// TIA Portal V18 export
DATA_BLOCK "Timers_DB"   // DB21
// stored: AutoNumber false, InstanceOfName Timers, InstanceOfType FB
"Timers"
   // VAR
   //    TDTimeReset : Bool;
   //    M1TimeReset : Bool;
   //    M2TimeReset : Bool;
   //    AuxTimeReset : Bool;
   //    CoolerTimeReset : Bool;
   //    TDRuntime : "Runtime_Out";
   //    M1Runtime { S7_SetPoint := 'True'} : "Runtime_Out";
   //    M2Runtime { S7_SetPoint := 'True'} : "Runtime_Out";
   //    AuxRuntime { S7_SetPoint := 'True'} : "Runtime_Out";
   //    CoolerRuntime { S7_SetPoint := 'True'} : "Runtime_Out";
   //    SystemRunStart : Bool;
   //    System_Runtime { S7_SetPoint := 'True'} : "Runtime";
   //    M1_Runtime { S7_SetPoint := 'True'} : "Runtime";
   //    M2_Runtime { S7_SetPoint := 'True'} : "Runtime";
   //    Cooler_Runtime { S7_SetPoint := 'True'} : "Runtime";
   //    AuxPump_Runtime { S7_SetPoint := 'True'} : "Runtime";
   // END_VAR
BEGIN
END_DATA_BLOCK
